// TIA Portal project "Proje1" (V15.1)

(* hardware
DEVICE "S7-1200 station_1"  S7-1200 Station
   slot 0: "Rack_0"  S7-1200 Rack  Rack  V1.0
   slot 1: "PLC_1"  CPU 1214C DC/DC/DC  6ES7 214-1AG40-0XB0  V4.2
DEVICE "HMI_1"  KTP700 Basic PN
   slot 0: "HMI_1"  KTP700 Basic PN  6AV2 123-2GB03-0AX0  15.1.0.0
   slot 1: "HMI_RT_1"  KTP700 Basic PN  6AV2 123-2GB03-0AX0  15.1.0.0
   slot 5: "HMI_1.IE_CP_1"  PROFINET Interface  15.0.1.0
      slot 1: "PROFINET Interface_1"  PROFINET Interface
         slot 1: "Port_1"  Port
*)

// ===== PLC "PLC_1"  CPU 1214C DC/DC/DC =====

VAR_GLOBAL   // PLC tag table "Default tag table"
   "System" AT %M0.0 : Bool;
   "Star contactor" AT %Q0.0 : Bool;
   "Delta contactor" AT %Q0.1 : Bool;
   "Insurance" AT %I0.0 : Bool;
   "Termik" AT %I0.1 : Bool;
   "Security" AT %M0.1 : Bool;
   "Start Time Reset" AT %M0.2 : Bool;
   "System_Byte" AT %MB1 : Byte;
   "FirstScan" AT %M1.0 : Bool;
   "DiagStatusUpdate" AT %M1.1 : Bool;
   "AlwaysTRUE" AT %M1.2 : Bool;
   "AlwaysFALSE" AT %M1.3 : Bool;
   "clockwise" AT %M0.3 : Bool;
   "counter clockwise" AT %M0.4 : Bool;
   "Direction contactor" AT %Q0.2 : Bool;
   "Direction Controller" AT %M0.5 : Bool;
   "Direction info" AT %M0.6 : Bool;
END_VAR

VAR_GLOBAL   // PLC tag table "Scl_Tag"
   "Start" AT %I0.2 : Bool;
   "Stop" AT %I0.3 : Bool;
   "Motor" AT %I0.4 : Bool;
END_VAR

DATA_BLOCK "Hmi_db"   // DB1
{ S7_Optimized_Access := 'TRUE' }
VERSION : 0.1
   VAR
      "Emergency Stop" : Bool;
      Restart : Bool;
      "Direction Reset" : Bool;
      Start : Bool;
      Stop : Bool;
      Star : Bool;
      Delta : Bool;
      "Elapsed Time Display" : Time;
      "Elapsed Time" : Time;
      "Selected Time" : Time := T#4ms;
      PT_Second : Time;
      clockwise : Bool;
      "counter clockwise" : Bool;
      "counter clockwise info" : Bool;
      "clockwise info" : Bool;
      "New PT" : Time := T#4ms;
   END_VAR
BEGIN
END_DATA_BLOCK

DATA_BLOCK "Csharp"   // DB3
{ S7_Optimized_Access := 'FALSE' }
VERSION : 0.1
   VAR
      "bit 1" : Bool;
   END_VAR
BEGIN
END_DATA_BLOCK

// folder: System blocks/Program resources

DATA_BLOCK "TP_timer"   // DB2
{ S7_Optimized_Access := 'TRUE' }
AUTHOR : Simatic
FAMILY : IEC
NAME : IEC_TMR
VERSION : 1.0
// stored: InstanceOfName IEC_TIMER
"IEC_TIMER"
BEGIN
END_DATA_BLOCK

// folder: (top level)

ORGANIZATION_BLOCK "Main"   // OB1, LAD, ProgramCycle
TITLE = "Main Program Sweep (Cycle)"
{ S7_Optimized_Access := 'TRUE' }
VERSION : 0.1
// Protection
   VAR_INPUT
      Initial_Call : Bool;   // Initial call of this OB
      Remanence : Bool;   // =True, if remanent data are available
   END_VAR
BEGIN

REGION Network 1
   // Termik and Insurance
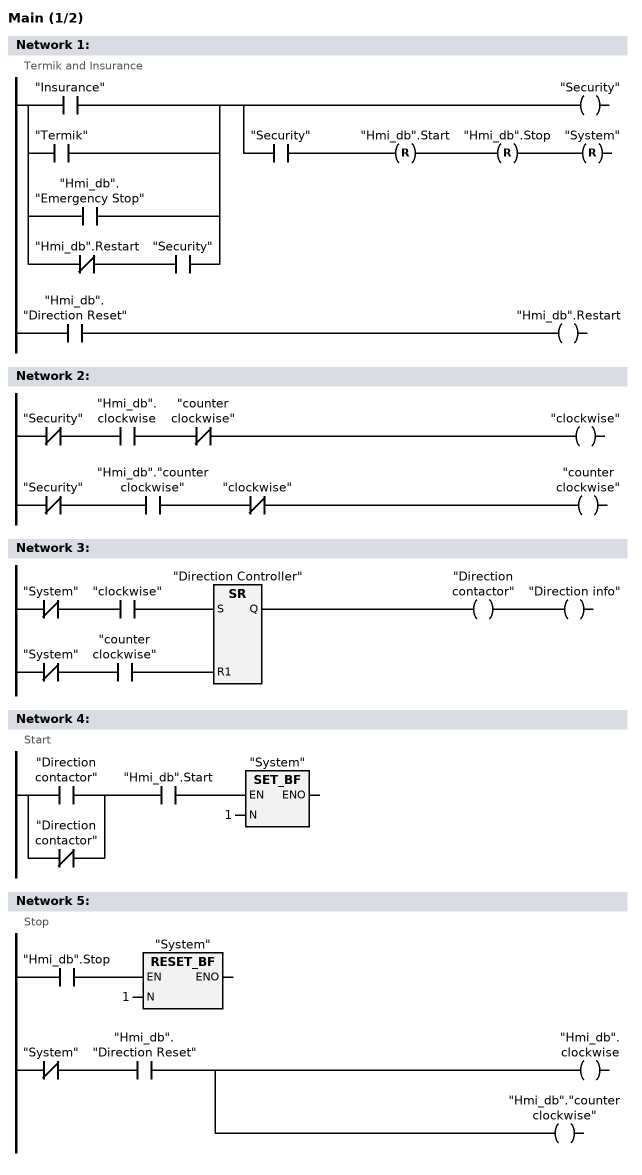
   RUNG wire#powerrail
      Contact( "Insurance" )
      wire#w1
      Coil( "Security" )
   END_RUNG
   RUNG wire#powerrail
      Contact( "Termik" )
   END_RUNG wire#w1
   RUNG wire#powerrail
      Contact( "Hmi_db"."Emergency Stop" )
   END_RUNG wire#w1
   RUNG wire#powerrail
      I_Contact( "Hmi_db".Restart )
      Contact( "Security" )
   END_RUNG wire#w1
   RUNG wire#w1
      Contact( "Security" )
      R_Coil( "Hmi_db".Start )
      R_Coil( "Hmi_db".Stop )
      R_Coil( "System" )
   END_RUNG
   RUNG wire#powerrail
      Contact( "Hmi_db"."Direction Reset" )
      Coil( "Hmi_db".Restart )
   END_RUNG
   // the same network as SCL:
   "Security" := "Insurance" OR "Termik" OR "Hmi_db"."Emergency Stop" OR (NOT "Hmi_db".Restart AND "Security");
   IF "Security" AND "Security" THEN
       "Hmi_db".Start := FALSE;
       "Hmi_db".Stop := FALSE;
       "System" := FALSE;
   END_IF;
   "Hmi_db".Restart := "Hmi_db"."Direction Reset";
END_REGION

REGION Network 2
   RUNG wire#powerrail
      I_Contact( "Security" )
      Contact( "Hmi_db".clockwise )
      I_Contact( "counter clockwise" )
      Coil( "clockwise" )
   END_RUNG
   RUNG wire#powerrail
      I_Contact( "Security" )
      Contact( "Hmi_db"."counter clockwise" )
      I_Contact( "clockwise" )
      Coil( "counter clockwise" )
   END_RUNG
   // the same network as SCL:
   "clockwise" := NOT "Security" AND "Hmi_db".clockwise AND NOT "counter clockwise";
   "counter clockwise" := NOT "Security" AND "Hmi_db"."counter clockwise" AND NOT "clockwise";
END_REGION

REGION Network 3
   RUNG wire#powerrail
      I_Contact( "System" )
      Contact( "clockwise" )
      S_SR(operand := "Direction Controller", r1 := wire#w1)
      Coil( "Direction contactor" )
      Coil( "Direction info" )
   END_RUNG
   RUNG wire#powerrail
      I_Contact( "System" )
      Contact( "counter clockwise" )
   END_RUNG wire#w1
   // the same network as SCL:
   IF NOT "System" AND "clockwise" THEN
       "Direction Controller" := TRUE;   // SR flip-flop
   END_IF;
   IF NOT "System" AND "counter clockwise" THEN "Direction Controller" := FALSE; END_IF;
   "Direction contactor" := "Direction Controller";
   "Direction info" := "Direction Controller";
END_REGION

REGION Network 4
   // Start
   // no SCL statement known for SBitfield: written as a call
   IF ("Direction contactor" OR NOT "Direction contactor") AND "Hmi_db".Start THEN
       SET_BF(operand := "System", n := 1);
   END_IF;
END_REGION

REGION Network 5
   // Stop
   // no SCL statement known for RBitfield: written as a call
   IF "Hmi_db".Stop THEN RESET_BF(operand := "System", n := 1); END_IF;
   "Hmi_db".clockwise := NOT "System" AND "Hmi_db"."Direction Reset";
   "Hmi_db"."counter clockwise" := "Hmi_db".clockwise;
END_REGION

REGION Network 6
   // PT Input
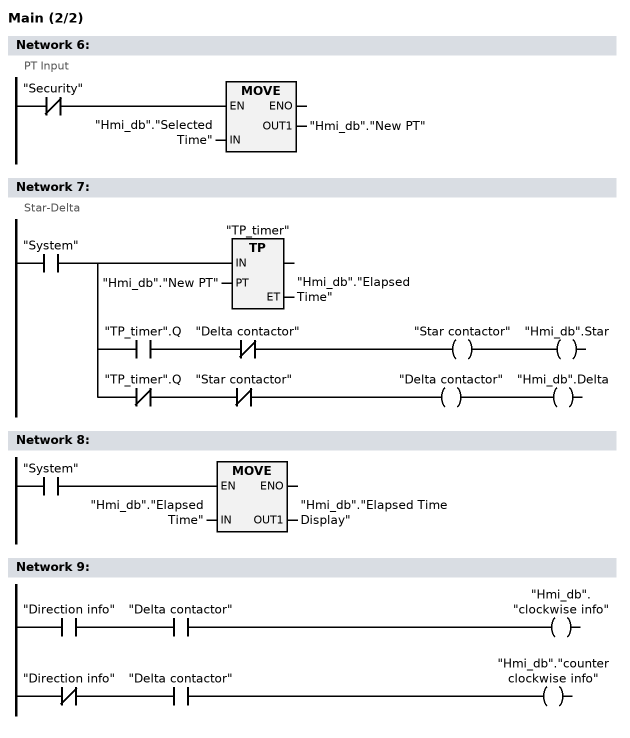
   RUNG wire#powerrail
      I_Contact( "Security" )
      Move(in := "Hmi_db"."Selected Time", out1 => "Hmi_db"."New PT")
   END_RUNG
   // the same network as SCL:
   IF NOT "Security" THEN "Hmi_db"."New PT" := "Hmi_db"."Selected Time"; END_IF;
END_REGION

REGION Network 7
   // Star-Delta
   "TP_timer".TP(IN := "System", PT := "Hmi_db"."New PT", ET => "Hmi_db"."Elapsed Time");
   "Star contactor" := "System" AND "TP_timer".Q AND NOT "Delta contactor";
   "Hmi_db".Star := "Star contactor";
   "Delta contactor" := "System" AND NOT "TP_timer".Q AND NOT "Star contactor";
   "Hmi_db".Delta := "Delta contactor";
END_REGION

REGION Network 8
   RUNG wire#powerrail
      Contact( "System" )
      Move(in := "Hmi_db"."Elapsed Time", out1 => "Hmi_db"."Elapsed Time Display")
   END_RUNG
   // the same network as SCL:
   IF "System" THEN "Hmi_db"."Elapsed Time Display" := "Hmi_db"."Elapsed Time"; END_IF;
END_REGION

REGION Network 9
   RUNG wire#powerrail
      Contact( "Direction info" )
      Contact( "Delta contactor" )
      Coil( "Hmi_db"."clockwise info" )
   END_RUNG
   RUNG wire#powerrail
      I_Contact( "Direction info" )
      Contact( "Delta contactor" )
      Coil( "Hmi_db"."counter clockwise info" )
   END_RUNG
   // the same network as SCL:
   "Hmi_db"."clockwise info" := "Direction info" AND "Delta contactor";
   "Hmi_db"."counter clockwise info" := NOT "Direction info" AND "Delta contactor";
END_REGION
END_ORGANIZATION_BLOCK

ORGANIZATION_BLOCK "SCL_deneme"   // OB123, SCL, ProgramCycle
TITLE = "Main Program Sweep (Cycle)"
{ S7_Optimized_Access := 'TRUE' }
VERSION : 0.1
   VAR_INPUT
      Initial_Call : Bool;   // Initial call of this OB
      Remanence : Bool;   // =True, if remanent data are available
   END_VAR
BEGIN
END_ORGANIZATION_BLOCK

(* ===== HMI "HMI_RT_1" =====
system functions are stored by id; their names below are inferred from use
connection "HMI_Connection_1": ETHERNET, SMART_S7_1200_OMS

HMI tags "Default tag table"
   "Tag_ScreenNumber" : UInt, internal
   "Hmi_db_Start" : Bool = PLC Hmi_db.Start, 100 ms
   "Hmi_db_Stop" : Bool = PLC Hmi_db.Stop, 100 ms
   "Hmi_db_Elapsed Time" : Time = PLC Hmi_db."Elapsed Time", 100 ms
   "Hmi_db_Selected Time" : Time = PLC Hmi_db."Selected Time", 1 s
   "Hmi_db_Star" : Bool = PLC Hmi_db.Star, 100 ms
   "Hmi_db_Delta" : Bool = PLC Hmi_db.Delta, 1 s
   "Hmi_db_clockwise" : Bool = PLC Hmi_db.clockwise, 1 s
   "Hmi_db_counter clockwise" : Bool = PLC Hmi_db."counter clockwise", 1 s
   "Hmi_db_clockwise info" : Bool = PLC Hmi_db."clockwise info", 1 s
   "Hmi_db_counter clockwise info" : Bool = PLC Hmi_db."counter clockwise info", 1 s
   "Hmi_db_Direction Reset" : Bool = PLC Hmi_db."Direction Reset", 1 s
   "Hmi_db_Emergency Stop" : Bool = PLC Hmi_db."Emergency Stop", 1 s
   "Direction info" : Bool = PLC "Direction info" AT %M0.6, 1 s
   "System" : Bool = PLC System AT %M0.0, 1 s
   "Security" : Bool = PLC Security AT %M0.1, 500 ms
   "Hmi_db_Elapsed Time Display" : Time = PLC Hmi_db."Elapsed Time Display", 1 s

HMI tags "Tag table_1"
   "Alarm" : Int, internal
   "Alarm-2" : Int, internal

discrete alarms
   1: 'Pressed run... / Çalıştır'a Basıldı...', class Errors, trigger "Alarm" bit 0
   2: 'Emergency Stop Status / Acil Stop Durumu', class Errors, trigger "Alarm-2" bit 1

graphic list "@DiagnosticsStates": 0 '@Diagnostics_StateGood'; 1 '@Diagnostics_StateBad'

Template "Main Template" 800x480
   Button "Exit" at 714,429 size 71x50; TextOff 'Exit'; PictureOn "ExitRuntime_KTP700_Basic_PN_TR"; PictureOff "Close-icon"
      on Release: StopRuntime(0)
      on Press: function_b14e0dd5("Hmi_db_Stop", 0)
   Button "Start screen" at 14,429 size 71x50; TextOff 'Text'; TextOn 'Start screen'; PictureOn "NavigateHome_KTP700_Basic_PN_TR"; PictureOff "home-icon"
      on Release: ActivateScreen("Main Menu", 0)
   DateTimeField "HmiScreenItemData" at 695,25 size 105x25
   DateTimeField "HmiScreenItemData_1" at 695,0 size 105x25
   GraphicView "Logo" at 0,0 size 109x51; Picture "Logo of HMI_1"
   Button "Start screen_1" at 154,430 size 71x50; TextOn 'Start screen'; TextOff 'Text'; PictureOn "NavigateHome_KTP700_Basic_PN_TR"; PictureOff "logout"; Authorization "User administration"
      on Release: ActivateScreen("User Login", 0); function_f23ef4c9()
   Button "Start screen_2" at 294,430 size 71x50; TextOff 'Text'; TextOn 'Start screen'; Authorization "User administration"; PictureOn "NavigateHome_KTP700_Basic_PN_TR"; PictureOff "Time-Date-To-icon"
      on Release: ActivateScreen("Alarm", 0)
   Button "Language_1" at 434,430 size 71x50; TextOn 'Language'; TextOff 'Language'; PictureOn "ToggleLanguage_KTP700_Basic_PN_TR"; PictureOff "Graphic_10"
      on Release: function_fb9197e8(L tr-TR)
   Button "Language_2" at 574,430 size 71x50; TextOn 'Language'; TextOff 'Language'; PictureOn "ToggleLanguage_KTP700_Basic_PN_TR"; PictureOff "Graphic_11"
      on Release: function_fb9197e8(L en-US)

screen "Main Menu" 800x480, template "Main Template"
   on GenerateScreen: SetTag("Tag_ScreenNumber", 1)
   Button "Button_1" at 270,143 size 102x62; TextOff 'START / Çalıştır'
      on Press: function_b14e0dd5("Hmi_db_Start", 0)
      on Release: function_b3f726e6("Alarm", 0)
   Button "Button_2" at 400,143 size 102x62; TextOff 'STOP / Durdur'
      on Press: function_b14e0dd5("Hmi_db_Stop", 0)
   IOField "I/O field_1" at 540,173 size 96x32; FormatPattern s9999999999
      ProcessValue <- "Hmi_db_Elapsed Time Display"
   TextField "Text field_1" at 536,145 size 68x23; Text 'Second / Saniye'
   IOField "I/O field_2" at 270,290 size 102x35; FormatPattern 99999
      ProcessValue <- "Hmi_db_Selected Time"
   TextField "Text field_3" at 175,239 size 435x23; Text 'Enter a value in seconds to change the star runtime / Yıldız çalışma süresini giriniz'
   Circle "Circle_1" at 660,145 size 71x71
      Appearance <- "Hmi_db_Star"
      Visibility <- "Hmi_db_Delta"
   TextField "Text field_4" at 176,290 size 69x42; Text 'Star Value Yıldız Değeri'
   TextField "Text field_5" at 428,364 size 16x23; Text 'Text'
   TextField "Text field_6" at 221,370 size 384x23; Text 'Motor running clockwise in delta connection / Motor saat yönünde üçgen bağlantıda çalışıyor'
      Visibility <- "Hmi_db_clockwise info"
   Button "Button_3" at 11,145 size 147x62; TextOff 'Clockwise / Saat Yönü'
      on Click: SetBit("Hmi_db_clockwise")
      Appearance <- "Direction info"
   Button "Button_5" at 11,223 size 149x62; TextOff 'Counter Clockwise / Saat Yönü Tersi'
      on Click: SetBit("Hmi_db_counter clockwise")
      Appearance <- "Direction info"
   TextField "Text field_2" at 194,370 size 430x23; Text 'Motor running counter clockwise in delta connection / Motor saat yönü tersinde üçgen bağlantıda çalışıyor'
      Visibility <- "Hmi_db_counter clockwise info"
   TextField "Text field_7" at 240,47 size 319x34; Text 'Asynchronous Motor Control / Asenkron Motor Kontrolü'
   Circle "Circle_2" at 660,145 size 71x71
      Appearance <- "Hmi_db_Delta"
      Visibility <- "Hmi_db_Star"
   GraphicView "Graphic view_1" at 11,78 size 54x57; Picture "reset"
   GraphicView "Graphic view_3" at 518,293 size 85x80; Picture "R_1"
      Visibility <- "Hmi_db_Star"
   GraphicView "Graphic view_2" at 523,273 size 110x91; Picture "delta"
      Visibility <- "Hmi_db_Delta"
   GraphicView "Graphic view_4" at 571,18 size 116x109; Picture "cross"
      Visibility <- "Security"
      Appearance <- "Security"
   Button "Button_4" at 0,78 size 86x55; TextOff 'Text'
      on Press: function_b14e0dd5("Hmi_db_Direction Reset", 0)
   Button "Button_6" at 84,78 size 69x55; TextOff 'Text'; PictureOff "Pushbutton_Emergency_On_256c"
      on Press: function_b14e0dd5("Hmi_db_Emergency Stop", 0); ActivateScreen("Alarm", 0); function_b3f726e6("Alarm-2", 1)

screen "User Login" 800x480, template "Login Template"
   Button "Button_1" at 9,167 size 131x65; TextOff 'Login / Giriş'; Authorization "User administration"
      on Release: ActivateScreen("Main Menu", 0)
   GraphicView "Graphic view_3" at 306,198 size 36x30; Picture "Graphic_8"
   GraphicView "Graphic view_4" at 398,206 size 36x30; Picture "Graphic_9"
   GraphicView "Graphic view_9" at 250,145 size 340x186; Picture "Graphic_14"
   TextField "Text field_1" at 306,45 size 16x23; Text 'Text'
   TextField "Text field_2" at 175,79 size 529x27; Text 'Welcome to the Asynchronous Motor Control Interface / Asenkron Motor Kontrolü Arayüzüne Hoşgeldiniz'

Template "Login Template" 800x480
   GraphicView "Logo" at 0,0 size 109x51; Picture "Logo of HMI_1"
   DateTimeField "HmiScreenItemData" at 695,25 size 105x25
   DateTimeField "HmiScreenItemData_1" at 695,0 size 105x25
   Button "Exit" at 714,429 size 71x50; TextOn 'Exit'; TextOff 'Exit'; PictureOn "ExitRuntime_KTP700_Basic_PN_TR"; PictureOff "Close-icon"
      on Release: StopRuntime(0)
      on Press: function_b14e0dd5("Hmi_db_Stop", 0)
   Button "Language_1" at 0,429 size 71x50; TextOn 'Language'; TextOff 'Language'; PictureOn "ToggleLanguage_KTP700_Basic_PN_TR"; PictureOff "Graphic_10"
      on Release: function_fb9197e8(L tr-TR)
   Button "Language_2" at 71,429 size 71x50; TextOn 'Language'; TextOff 'Language'; PictureOn "ToggleLanguage_KTP700_Basic_PN_TR"; PictureOff "Graphic_11"
      on Release: function_fb9197e8(L en-US)

screen "Alarm" 800x480, template "Main Template"
   AlarmView "Alarm view_1" at 68,120 size 651x300
   Button "Button_1" at 715,61 size 79x56; TextOff 'Text'; PictureOff "return"
      on Release: ActivateScreen("Main Menu", 0)
*)